FUNCTION_BLOCK FB_BrakeTorque
VAR_INPUT
	
	iTorqueValueinNm: INT;
END_VAR

VAR_OUTPUT
	iTorqueScaled: INT; //Scaled torque value 
    
END_VAR
	
VAR
	iTorqueMin:INT := 2; // Min brake torque in Nm
	iTorqueMax:INT := 200; // Max brake torque in Nm
	iVoltageDecMin:INT := 0; // 0V in decimal representation
	iVoltageDecMax:INT := 32767; //10V in decimal representation

END_VAR

IF iTorqueValueinNm >=2 THEN

iTorqueScaled := ((iTorqueValueinNm-iTorqueMin)/(iTorqueMax-iTorqueMin))*(iVoltageDecMax-iVoltageDecMin) + iVoltageDecMin;
//Global_IO.iqAnalogueOut_1:=iTorqueScaled;

END_IF

END_FUNCTION_BLOCK

(* stored: Version 1.1.0.1, ProductVersion 3.1.4022.10
   POU FB_BrakeTorque: Id {ac54a68e-0c0d-4c2e-a105-bba2ce4e7751}, SpecialFunc None *)
